// Copyright (c) 2024 Loupe (https://loupe.team), provided under the MIT License.
TYPE AbbLinkinRequestQueue_Typ :
STRUCT
	request : AbbLinkinRequest_Typ;
	empty : BOOL := TRUE;
END_STRUCT
END_TYPE

(* stored: Version 1.1.0.1, ProductVersion 3.1.4024.12
   DUT AbbLinkinRequestQueue_Typ: Id {0da73142-5815-463c-9973-c8dbb7228de0} *)
